(*********************************** G.D S.p.A. - Technical Department ***********************************
============= PROGRAM INFO ============
FOLDER:             TBD
MACHINES INVOLVED:  TBD 

============= DESCRIPTION =============
Low task

============= REVISIONS ===============
Date		Version	 	Author      	Description             
----------	-------		------------  	--------------------------------------------
2019/03/28 	0000.00	 	CEC		 		Creation of the PRG

**********************************************************************************************************)

PROGRAM _csp_customerInterfaces_normal
VAR
END_VAR

;

END_PROGRAM

(* stored: Version 1.1.0.1, ProductVersion 3.1.4022.12
   POU _csp_customerInterfaces_normal: Id {3cb04ded-0371-4a7a-a320-3d868fc82db0}, SpecialFunc None *)
